FUNCTION F_GetConnectionString : STRING
VAR_INPUT
    bConnected : BOOL;
END_VAR
VAR
END_VAR

IF bConnected THEN
    F_GetConnectionString := 'Connected';
ELSE
    F_GetConnectionString := 'Disconnected';
END_IF

END_FUNCTION

(* stored: Version 1.1.0.1, ProductVersion 3.1.4024.14
   POU F_GetConnectionString: Id {c38a4031-5dde-420b-9d0c-d82ada4d6489}, SpecialFunc None *)
